{attribute addProperty BoxType "EK1960-0000-0019"}
{attribute addProperty Id "FSOEAT %Q*FSOE_B1AE0A9412015"}
{attribute addProperty CRC "2468202949"}
{attribute addProperty SizeInBites "120"}
{attribute addProperty SizeInBytes "15"}
TYPE FSoE_Outputs_931DC9C5 :
STRUCT
	{attribute addProperty Name "FSOE"}
	FSOE AT %Q* : FSOE_B1AE0A94;
END_STRUCT
END_TYPE

(* stored: Version 1.2.0.0, ProductVersion 3.1.4024.9
   DUT FSoE_Outputs_931DC9C5: Id {2a861863-a132-494a-b8ad-de6675c62a48} *)
